FUNCTION UPPERCASE : STRING(STRING_LENGTH)
VAR_INPUT
	str : STRING(STRING_LENGTH);
END_VAR
VAR
	pt : POINTER TO BYTE;
	pos: INT;
	l: INT;
END_VAR

(*
version 1.3	29. mar. 2008
programmer 	hugo
tested by	tobias

uppercase returns str while all letters a..z and ä,ö,ü are converted to uppercase

*)

pt := ADR(UPPERCASE);
UPPERCASE := str;
l := LEN(str);
FOR pos := 1 TO l DO
	pt^ := TO_UPPER(pt^);
	pt := pt + 1;
END_FOR;

(* revision histroy
hm	6. oct. 2006	rev 1.0
	original release

hm	4. feb. 2008	rev 1.1
	improved performance
	added Ä,Ö,Ü

hm	6. mar. 2008	rev 1.2
	added support for exteded Ascii

hm	29. mar. 2008	rev 1.3
	changed STRING to STRING(STRING_LENGTH)

*)

END_FUNCTION

(* stored: Version 1.1.0.1, ProductVersion 3.1.4022.7
   POU UPPERCASE: Id {fc9b7e98-9df1-455c-b4e3-12621d8745cc}, SpecialFunc None *)
